PROGRAM AxisReset
VAR

END_VAR

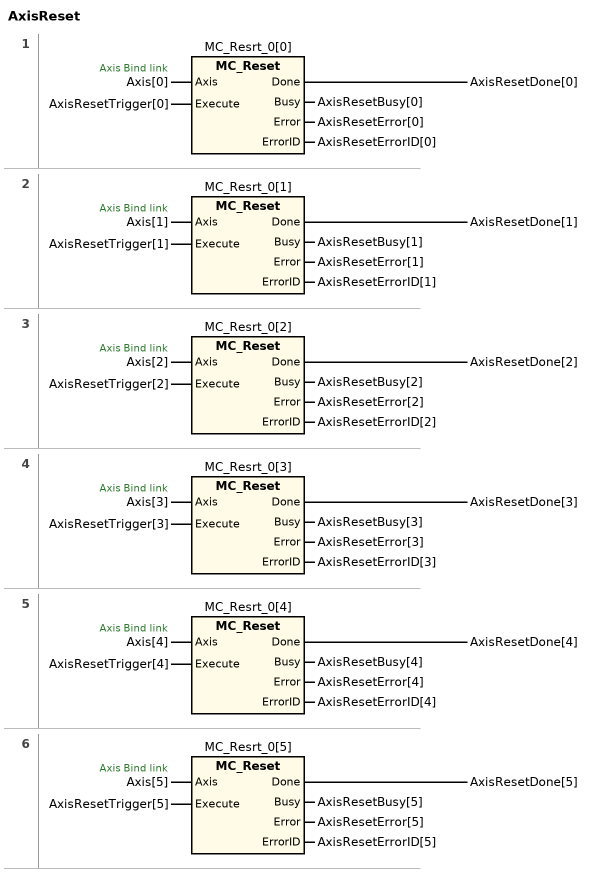
// NETWORK 1
//   MC_Resrt_0[0]: Reset
//   Axis[0]: Axis Bind link
MC_Resrt_0[0](
    Axis := Axis[0],
    Execute := AxisResetTrigger[0],
    Busy => AxisResetBusy[0],
    Error => AxisResetError[0],
    ErrorID => AxisResetErrorID[0]); // MC_Reset
AxisResetDone[0] := MC_Resrt_0[0].Done;

// NETWORK 2
//   MC_Resrt_0[1]: Reset
//   Axis[1]: Axis Bind link
MC_Resrt_0[1](
    Axis := Axis[1],
    Execute := AxisResetTrigger[1],
    Busy => AxisResetBusy[1],
    Error => AxisResetError[1],
    ErrorID => AxisResetErrorID[1]); // MC_Reset
AxisResetDone[1] := MC_Resrt_0[1].Done;

// NETWORK 3
//   MC_Resrt_0[2]: Reset
//   Axis[2]: Axis Bind link
MC_Resrt_0[2](
    Axis := Axis[2],
    Execute := AxisResetTrigger[2],
    Busy => AxisResetBusy[2],
    Error => AxisResetError[2],
    ErrorID => AxisResetErrorID[2]); // MC_Reset
AxisResetDone[2] := MC_Resrt_0[2].Done;

// NETWORK 4
//   MC_Resrt_0[3]: Reset
//   Axis[3]: Axis Bind link
MC_Resrt_0[3](
    Axis := Axis[3],
    Execute := AxisResetTrigger[3],
    Busy => AxisResetBusy[3],
    Error => AxisResetError[3],
    ErrorID => AxisResetErrorID[3]); // MC_Reset
AxisResetDone[3] := MC_Resrt_0[3].Done;

// NETWORK 5
//   MC_Resrt_0[4]: Reset
//   Axis[4]: Axis Bind link
MC_Resrt_0[4](
    Axis := Axis[4],
    Execute := AxisResetTrigger[4],
    Busy => AxisResetBusy[4],
    Error => AxisResetError[4],
    ErrorID => AxisResetErrorID[4]); // MC_Reset
AxisResetDone[4] := MC_Resrt_0[4].Done;

// NETWORK 6
//   MC_Resrt_0[5]: Reset
//   Axis[5]: Axis Bind link
MC_Resrt_0[5](
    Axis := Axis[5],
    Execute := AxisResetTrigger[5],
    Busy => AxisResetBusy[5],
    Error => AxisResetError[5],
    ErrorID => AxisResetErrorID[5]); // MC_Reset
AxisResetDone[5] := MC_Resrt_0[5].Done;

END_PROGRAM

(* stored: Version 1.1.0.1, ProductVersion 3.1.4018.5
   POU AxisReset: Id {6839d459-e108-4514-878a-73b7c3033a0c}, SpecialFunc None *)
